VAR_GLOBAL CONSTANT
	nInitialize: SINT := 0;
	nStep: SINT := 1;
END_VAR

(* stored: Version 1.1.0.1, ProductVersion 3.1.4024.9
   GVL GVL_PID: Id {dfa854b2-a47f-4123-a810-d4207c26d488} *)
